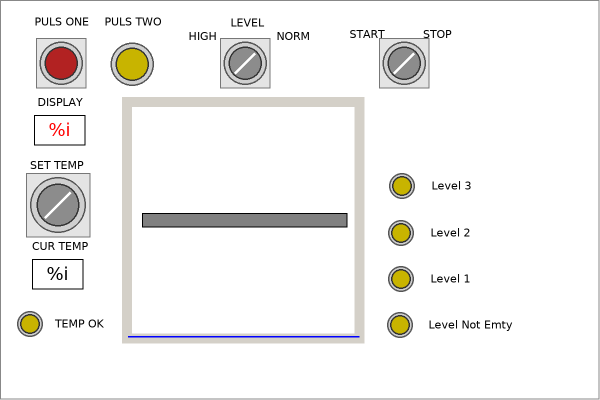
VISUALIZATION Visualization  // 600x400
    Rectangle (122,97 242x246)
    PushSwitch (36,38 50x50), variable: GVL.qxPulseOne, behaviour: TOGGLE, style: Switch-PushSwitch-Red
    Label (10,11 104x22), "PULS ONE"
    RotarySwitch (220,38 50x50), variable: GVL.qxSetLevel, input disabled if: GVL.qxStart, behaviour: TOGGLE, style: Switch-RotarySwitch-Gray
    Label (164,10 160x39), "LEVEL HIGH NORM"
    RotarySwitch (379,38 50x50), variable: GVL.qxStart, behaviour: TOGGLE, style: Switch-RotarySwitch-Gray
    Label (317,15 160x39), "START STOP"
    Lamp1 (387,171 30x30), variable: GVL.qxLevel3, style: Lamp-Lamp1-Yellow
    Label (420,178 63x16), "Level 3"
    Lamp1 (386,218 30x30), variable: GVL.qxLevel2, style: Lamp-Lamp1-Yellow
    Label (419,225 63x16), "Level 2"
    Lamp1 (386,264 30x30), variable: GVL.qxLevel1, style: Lamp-Lamp1-Yellow
    Label (419,271 63x16), "Level 1"
    Lamp1 (385,310 30x30), variable: GVL.qxNotEmpty, style: Lamp-Lamp1-Yellow
    Label (418,317 105x16), "Level Not Emty"
    Lamp1 (15,309 30x30), variable: GVL.qxTempOk, style: Lamp-Lamp1-Yellow
    Label (48,316 63x16), "TEMP OK"
    Potentiometer360 (24,173 68x64), variable: GVL.qwSetTem, style: Potentiometer-Potentiometer360-Gray, scale format: %i, scale 0..100
        p2431819421: Outside
    Rectangle (32,259 51x30), "%i", text variable: GVL.qwCurTemp
    Label (14,237 92x19), "CUR TEMP"
    Label (11,156 92x19), "SET TEMP"
    Label (14,93 92x19), "DISPLAY"
    Rectangle (34,115 51x30), "%i", text variable: GVL.qwSetTem
    Rectangle (128,336 231x1)
        p2773130477: GVL.nShowWater
    Rectangle (142,213 205x14)
        p2858320360: GVL.nCylPos
    Label (81,11 104x22), "PULS TWO"
    Lamp1 (107,39 50x50), variable: GVL.ixPulseTwo, style: Lamp-Lamp1-Yellow
END_VISUALIZATION

(* stored: Version 1.1.0.1, ProductVersion 3.1.4024.12
   Visu Visualization: Id {ad45f26b-89f6-408d-b081-64ca21bca6cc} *)
